{attribute 'qualified_only'}
VAR_GLOBAL

	//Internal powermeter variables	
	Power_analyzer: 			Meter_board_str;
	Meter_comms_status: 		BOOL;
	
	//Internal calculated powermeter variables
		//Average voltages in engineering units
	V_phase_avg_Volt:			REAL;
	V_line_avg_Volt:			REAL;
		//Single-phase electrical parameters in p.u.
	P_L1_pu:					REAL;
	P_L2_pu:					REAL;
	P_L3_pu:					REAL;
	Q_L1_pu:					REAL;
	Q_L2_pu:					REAL;
	Q_L3_pu:					REAL;
	S_L1_pu:					REAL;
	S_L2_pu:					REAL;
	S_L3_pu:					REAL;
	V_L1N_pu:					REAL;
	V_L2N_pu:					REAL;
	V_L3N_pu:					REAL;
	I_L1_pu:					REAL;
	I_L2_pu:					REAL;
	I_L3_pu:					REAL;
		//Three-phase electrical parameters in p.u.
	P_pu:						REAL;
	Q_pu:						REAL;
	S_pu:						REAL;
		//Average voltages in engineering units
	V_phase_avg_pu:				REAL;
	V_line_avg_pu:				REAL;
	
	//Self-supply P variables
	P_min:						REAL; //Minimum P in p.u. of the system for PI feedback
	P_min_indicator:			WORD; //Minimum P indicator 0 --> L1; 1 --> L2; 2 --> L3

	//Enrgies handling & values
	Energies_reset:				BOOL:= FALSE;
	Active_er_neg_kWh: 			LINT:=0; //Active energy (three-phase) calculated if P_tot < 0
	Active_er_pos_kWh:			LINT:=0; //Active energy (three-phase) calculated if P_tot > 0
	Active_er_tot_kWh: 			LINT:=0; //Active energy (three-phase) calculated. Net calculation
	React_er_neg_kVArh: 		LINT:=0; //Rective energy (three-phase) calculated if Q_tot < 0
	React_er_pos_kVArh: 		LINT:=0; //Rective energy (three-phase) calculated if Q_tot > 0
	React_er_tot_kVArh: 		LINT:=0; //Reactive energy (three-phase) calculated. Net calculation
	
	//Data to be linked to metering board
	//Single-phase data
	M_board_P_L1_kW				AT %I*	: REAL;
	M_board_P_L2_kW				AT %I*	: REAL;		
	M_board_P_L3_kW				AT %I*	: REAL;		
	M_board_Q_L1_kVAr			AT %I*	: REAL;		
	M_board_Q_L2_kVAr			AT %I*	: REAL;		
	M_board_Q_L3_kVAr			AT %I*	: REAL;		
	M_board_S_L1_kVA			AT %I*	: REAL;		
	M_board_S_L2_kVA			AT %I*	: REAL;		
	M_board_S_L3_kVA			AT %I*	: REAL;		
	M_board_cos_phi_L1			AT %I*	: REAL;		
	M_board_cos_phi_L2			AT %I*	: REAL;		
	M_board_cos_phi_L3			AT %I*	: REAL;		
	M_board_V_L1N_Volt			AT %I*	: REAL;		
	M_board_V_L2N_Volt			AT %I*	: REAL;		
	M_board_V_L3N_Volt			AT %I*	: REAL;					
						
	//Three-phase data			
	M_board_P_kW				AT %I*	: REAL;	
	M_board_Q_kVAr				AT %I*	: REAL;	
	M_board_S_kVA				AT %I*	: REAL;	
	M_board_Freq_Hz				AT %I*	: REAL;		
	M_board_cos_phi				AT %I*	: REAL;		
	M_board_V_L1L2_Volt			AT %I*	: REAL;			
	M_board_V_L2L3_Volt			AT %I*	: REAL;			
	M_board_V_L3L1_Volt			AT %I*	: REAL;			
	M_board_I_L1_angle			AT %I*	: REAL;		
	M_board_I_L2_angle			AT %I*	: REAL;		
	M_board_I_L3_angle			AT %I*	: REAL;		
	M_board_V_L1L2_angle		AT %I* 	: REAL;			
	M_board_V_L1L3_angle		AT %I*	: REAL;					
	
	//Rest of data								
	M_board_Meter_status		AT %I*	: WORD;
END_VAR

VAR_GLOBAL PERSISTENT
	Alg_lost_comms_enable: 		BOOL:= FALSE;
END_VAR

(* stored: Version 1.1.0.1, ProductVersion 3.1.4024.11
   GVL GVL_POWERMETER: Id {f138ff50-4403-486f-b4af-1f0f47357b23} *)
